FUNCTION_BLOCK Mc3MotionHomeTask_SetPosition EXTENDS Mc3MotionTask
VAR
	MCSetPosition : Tc3_Mc3Ptp.MC_SetPosition;
	_HomePosition : LREAL := 0.0;
END_VAR

{attribute 'monitoring' := 'call'}
PROPERTY Busy : BOOL
GET
Busy := MCSetPosition.Busy;
END_GET
END_PROPERTY

METHOD CyclicLogic
MCSetPosition(Axis := _Axis.Axis, Position := HomePosition);
MCSetPosition.Execute := FALSE;
END_METHOD

{attribute 'monitoring' := 'call'}
PROPERTY Error : BOOL
GET
Error := MCSetPosition.Error;
END_GET
END_PROPERTY

{attribute 'monitoring' := 'call'}
PROPERTY ErrorId : UDINT
GET
ErrorId := MCSetPosition.ErrorID;
END_GET
END_PROPERTY

METHOD Execute : BOOL
IF Axis.Busy OR Axis.Error THEN
	RETURN;
END_IF

MCSetPosition.Execute := TRUE;
Execute				  := TRUE;
END_METHOD

PROPERTY HomePosition : LREAL
GET
HomePosition := MCSetPosition.Position;
END_GET
SET
MCSetPosition.Position := HomePosition;
END_SET
END_PROPERTY

END_FUNCTION_BLOCK

(* stored: Version 1.1.0.1, ProductVersion 3.1.4026.20
   POU Mc3MotionHomeTask_SetPosition: Id {d3b78bba-a9ad-4679-92bf-b0571a9c2764}, SpecialFunc None
   Property Busy: Id {0de1f59a-f835-4223-9285-45fd155f6776}
   Get Get: Id {fd7221c9-0829-4102-8be6-e559bf34b3e2}
   Method CyclicLogic: Id {095145ce-0a46-448d-bb7d-9b71043631a0}
   Property Error: Id {4514c2a9-4766-4df4-a1dd-7fcda466c142}
   Get Get: Id {d3b6d3dc-aeec-407b-91db-d02b0102e6e7}
   Property ErrorId: Id {e4314d5a-f850-4bbf-a7f9-ddfc07b44edb}
   Get Get: Id {e0e8922b-d7cf-41a5-880f-f8a691747989}
   Method Execute: Id {5a4245c8-7389-4372-925d-218c7a9f0262}
   Property HomePosition: Id {4693e885-e1f1-4fa7-983c-d58caa539bb3}
   Get Get: Id {30bf28d0-206c-4c07-a45f-1ea554d4b85f}
   Set Set: Id {48bda34a-1dba-474d-9f2d-44952a76b527} *)
